{attribute 'linkalways'} 
{attribute 'no_explicit_call' := 'This FB is a CLASS and must be accessed using methods or properties'}
{attribute 'enable_dynamic_creation'}
FUNCTION_BLOCK Node_F_VN_GetRoi EXTENDS VisionNode
VAR
    ipSrcImage : _ITcVnImage;
    stRoi : _TcVnRectangle_UDINT;
    hrPrev : _HRESULT(S_OK);
	hresult : _HRESULT(S_OK);
END_VAR

METHOD PUBLIC  Clone : I_Node
VAR
	pNode : POINTER TO Node_F_VN_GetRoi;
END_VAR
pNode := __NEW(Node_F_VN_GetRoi);
Clone := pNode^;
END_METHOD

METHOD FB_init : BOOL
VAR_INPUT
	bInitRetains : BOOL; // if TRUE, the retain variables are initialized (warm start / cold start)
	bInCopyCode : BOOL;  // if TRUE, the instance afterwards gets moved into the copy code (online change)
END_VAR
AddInput('ipSrcImage', ipSrcImage);
AddInput('hrPrev', hrPrev);
AddOutput('stRoi', stRoi);
AddOutput('hresult',hresult);
END_METHOD

METHOD PROTECTED  OnExecute : HRESULT
hresult.Value := F_VN_GetRoi(
    ipSrcImage := ipSrcImage.Value,
    stRoi := stRoi.Value,
	hrPrev:= hrPrev.Value);
END_METHOD

METHOD PUBLIC PreExecutionCheck
VAR_INPUT
	Check : I_PreExecutionChecks;
END_VAR
IF FAILED(hrPrev.Value) THEN
    RETURN;
END_IF

Check.IsTrue(ipSrcImage.IsValid, 'ipSrcImage must contain an image');
END_METHOD

END_FUNCTION_BLOCK

(* stored: Version 1.1.0.1, ProductVersion 3.1.4024.13
   POU Node_F_VN_GetRoi: Id {4752c226-55d5-0a48-3e98-2bf2ff30d83d}, SpecialFunc None
   Folder Constructor: Id {444d82fe-983b-0025-2ed1-970eafaef0ce}
   Method Clone: Id {73a5c906-35eb-0e28-0f26-3b6e93b383fb}
   Method FB_init: Id {75390258-63ba-03ed-39f7-b55493b7f381}
   Method OnExecute: Id {0c2b7e68-6b9a-069c-1968-53061b721031}
   Method PreExecutionCheck: Id {288aa9dd-63e5-0cb5-077c-3597ebd723f8} *)
